// TIA Portal V20 export
FUNCTION_BLOCK "FB_PartControl"   // FB58, SCL
{ S7_Optimized_Access := 'TRUE' }
// stored: MemoryReserve 100, SetENOAutomatically false
   VAR_INPUT
      iStartSeqCond : Bool;   // Start Sequence Conditions
      iJobReq : Bool;   // Job Request - From Main
      iCtrlEnabled : Bool;   // Part Control Enable - Param or Condition
      iShuttleCtrlUndrilledPos : Bool;   // Undrilled Pos. Reached (Option Individual Ctrl) - Param
      iShuttleCtrlUndrilledPosSetPoint : LReal;   // Undrilled Pos. Setpoint (Option Individual Ctrl) - Param
      iShuttleCtrlDrilledPos : Bool;   // Drilled Pos. Reached (Option Individual Ctrl) - Param
      iShuttleCtrlDrilledPosSetPoint : LReal;   // Drilled Pos. Setpoint (Option Individual Ctrl) - Param
      iShuttleCtrlPos : Bool;   // Control Pos. Reached (Option Common Ctrl) - Param
      iShuttleCtrlPosSetPoint : LReal;   // Control Pos. Setpoint (Option Common Ctrl) - Param
      iExpectedCtrlUndrilled : Bool;   // Expected result Undrilled Pos.
      iExpectedCtrlDrilled : Bool;   // Expected result Drilled Pos.
      iPartMeasureValue : Real;   // Part Measure Value (Option Analog Measure) - From AI
      iPartMeasureTolMin : Real;   // Part Tol Min Value (Option Analog Measure) - Param
      iPartMeasureTolMax : Real;   // Part Tol Max Value (Option Analog Measure) - Param
      iUndrilledPartPresence : Bool;
      iDrilledPartPresence : Bool;
      iShuttleMoving : Bool;   // Shuttle is moving - From FB_LoaderAxis
      iShuttleInPos : Bool;   // Shuttle pos. reached - From FB_LoaderAxis
      iPLC_DateAndTime : DTL;
      iStepPause : Bool;
   END_VAR
   VAR_OUTPUT
      oShuttleStartReq { ExternalAccessible := 'False'; ExternalVisible := 'False'; ExternalWritable := 'False'} : Bool;   // Shuttle Start Order - To FB_LoaderAxis
      oShuttlePosSetPoint { ExternalAccessible := 'False'; ExternalVisible := 'False'; ExternalWritable := 'False'} : Real;   // Shuttle Position Setpoint - To FB_LoaderAxis
      oPartControlOK : Bool;   // Part OK - To Main
      oPartControlNOK : Bool;   // Part NOK - To Main
   END_VAR
   VAR
      sCurrent_Step_NB : Int;   // Active Step Number
      sCheck_Step_Condition : Bool;
      sOneStepForward : Bool;
      sRTOneStepForward : R_TRIG;
      sOneStepMode { S7_SetPoint := 'True'} : Bool;
      sStepForward : Bool;
      sInterface : "UDT_SequenceInterface";
      sShuttleStartReq { ExternalAccessible := 'False'; ExternalVisible := 'False'; ExternalWritable := 'False'} : Bool;
      sShuttlePosSetPoint { ExternalAccessible := 'False'; ExternalVisible := 'False'; ExternalWritable := 'False'} : Real;
      sMissingPartCtrlUndrilled : Bool;
      sMissingPartCtrlDrilled : Bool;
      sExtraPartCtrlUndrilled : Bool;
      sExtraPartCtrlDrilled : Bool;
      sPresencePartUndrilledPos : Bool;
      sPresencePartDrilledPos : Bool;
      sPartControlOK : Bool;
      sPartControlNOK : Bool;
      sControlTimer : TON_TIME;
      sHistory : Struct
         Activation : Bool;
         Steps : Array[0..99] of Int;
         Date_Time : Array[0..99] of DTL;
      END_STRUCT;
      StepText : "FB_GetTextErrorCode";
   END_VAR
   VAR_TEMP
      tIndex : Int;   // Index
   END_VAR
   VAR CONSTANT
      S00_INIT : Int := 0;
      S10_CHECK_PART_PRESENCE_OPTION : Int := 10;
      S20_SHUTTLE_TO_UNDRILLED_POS_START_REQ : Int := 20;
      S30_SHUTTLE_TO_UNDRILLED_POS_REACHED : Int := 30;
      S40_WAIT_UNDRILLED_CTRL_EXECUTION : Int := 40;
      S50_SHUTTLE_TO_DRILLED_POS_START_REQ : Int := 50;
      S60_SHUTTLE_TO_DRILLED_POS_REACHED : Int := 60;
      S70_WAIT_DRILLED_CTRL_EXECUTION : Int := 70;
      S80_CHECK_PART_POS_RESULT : Int := 80;
      S120_SHUTTLE_TO_CONTROL_POS_START_REQ : Int := 120;
      S130_SHUTTLE_TO_CONTROL_POS_REACHED : Int := 130;
      S140_WAIT_CONTROL_EXECUTION : Int := 140;
      S180_CHECK_PART_POS_RESULT : Int := 180;
      S280_NO_PART_CTRL : Int := 280;
      S295_JOB_DONE : Int := 295;
   END_VAR
   // StepText.sCode_error[0].ErrorCode := 0;
   // StepText.sCode_error[1].ErrorCode := 10;
   // StepText.sCode_error[2].ErrorCode := 20;
   // StepText.sCode_error[3].ErrorCode := 30;
   // StepText.sCode_error[4].ErrorCode := 40;
   // StepText.sCode_error[5].ErrorCode := 50;
   // StepText.sCode_error[6].ErrorCode := 60;
   // StepText.sCode_error[7].ErrorCode := 70;
   // StepText.sCode_error[8].ErrorCode := 80;
   // StepText.sCode_error[9].ErrorCode := 90;
   // StepText.sCode_error[10].ErrorCode := 95;
BEGIN
   REGION Description header 
       //==================================================================================
       // POSALUX Swiss SA / (C) Copyright 2025
       //----------------------------------------------------------------------------------
       // Title: FB_PartControl
       // Comment/Function: 
       // Author: Fabien WALDT
       // Engineering: TIA Portal v17
       //----------------------------------------------------------------------------------
       // Change log table:
       // Version  | Date     | Expert in charge | Changes applied
       // ---------|----------|------------------|-----------------------------------------
       // 00.00.01 | 20250527 | WFA              | First released version
       // =================================================================================
   END_REGION

   REGION Define condition to start
       IF #iStartSeqCond THEN
           #sInterface.SequenceReleased := TRUE;
       ELSE
           // Standard sequencer controls
           #sInterface.SequenceReleased := FALSE;
           #sCurrent_Step_NB := #S00_INIT;
           #sInterface.SequenceRun := FALSE;
           #sInterface.JobDone := FALSE;
           #sCheck_Step_Condition := FALSE;

           // Dedicated sequencer controls
           #sShuttleStartReq := FALSE;
           #sShuttlePosSetPoint := 0.0;
           #sPresencePartUndrilledPos := FALSE;
           #sPresencePartDrilledPos := FALSE;

           // Add specifics controls 
       END_IF;

       // Reset interface error
       IF #sInterface.Reset THEN
           #sInterface.Error := FALSE;
       END_IF;

       // Reset start when axis in position
       IF #iShuttleInPos THEN
           #sShuttleStartReq := FALSE;
       END_IF;

       // One step forward
       #sRTOneStepForward.CLK := #sOneStepForward;
       #sRTOneStepForward();
       #sStepForward := (NOT #sOneStepMode OR (#sOneStepMode AND #sRTOneStepForward.Q)) AND NOT #iStepPause;
       #sOneStepForward := FALSE;

       // Step Timer
       #sControlTimer(IN := #sCurrent_Step_NB = 40 OR #sCurrent_Step_NB = 140,
                            PT := T#50ms);
   END_REGION

   REGION Sequence Function
       CASE #sCurrent_Step_NB OF
           #S00_INIT:
               REGION S00 INIT
                   #sCheck_Step_Condition := TRUE;
               END_REGION
           #S10_CHECK_PART_PRESENCE_OPTION:
               REGION S10_CHECK_PART_PRESENCE_OPTION
                   #sPartControlOK := FALSE;
                   #sPartControlNOK := FALSE;
                   #sMissingPartCtrlUndrilled := FALSE;
                   #sMissingPartCtrlDrilled := FALSE;
                   #sExtraPartCtrlUndrilled := FALSE;
                   #sExtraPartCtrlDrilled := FALSE;
                   #sCheck_Step_Condition := TRUE;
               END_REGION
           #S20_SHUTTLE_TO_UNDRILLED_POS_START_REQ:
               REGION S20_SHUTTLE_TO_UNDRILLED_POS_START_REQ
                   #sShuttleStartReq := NOT #iShuttleCtrlUndrilledPos;
                   #sShuttlePosSetPoint := LREAL_TO_REAL(#iShuttleCtrlUndrilledPosSetPoint);
                   #sCheck_Step_Condition := TRUE;
               END_REGION
           #S30_SHUTTLE_TO_UNDRILLED_POS_REACHED:
               REGION S30_SHUTTLE_TO_UNDRILLED_POS_REACHED
                   #sCheck_Step_Condition := TRUE;
               END_REGION
           #S40_WAIT_UNDRILLED_CTRL_EXECUTION:
               REGION S40_WAIT_UNDRILLED_CTRL_EXECUTION
                   IF "DB_LoaderOptions".PartControl.AnalogMeasure THEN
                       IF #iPartMeasureValue > #iPartMeasureTolMin AND #iPartMeasureValue < #iPartMeasureTolMax THEN
                           #sPresencePartUndrilledPos := TRUE;
                       ELSE
                           #sPresencePartUndrilledPos := FALSE;
                       END_IF;
                   ELSIF "DB_LoaderOptions".PartControl.DigitalMeasure THEN
                       IF #iUndrilledPartPresence THEN
                           #sPresencePartUndrilledPos := TRUE;
                       ELSE
                           #sPresencePartUndrilledPos := FALSE;
                       END_IF;
                       IF #iDrilledPartPresence THEN
                           #sPresencePartDrilledPos := TRUE;
                       ELSE
                           #sPresencePartDrilledPos := FALSE;
                       END_IF;
                   ELSE
                       #sInterface.Error := TRUE;
                   END_IF;
                   IF #sControlTimer.Q THEN
                       #sCheck_Step_Condition := TRUE;
                   END_IF;
               END_REGION
           #S50_SHUTTLE_TO_DRILLED_POS_START_REQ:
               REGION S50_SHUTTLE_TO_DRILLED_POS_START_REQ
                   #sShuttleStartReq := NOT #iShuttleCtrlDrilledPos;
                   #sShuttlePosSetPoint := LREAL_TO_REAL(#iShuttleCtrlDrilledPosSetPoint);
                   #sCheck_Step_Condition := TRUE;
               END_REGION
           #S60_SHUTTLE_TO_DRILLED_POS_REACHED:
               REGION S60_SHUTTLE_TO_DRILLED_POS_REACHED
                   #sCheck_Step_Condition := TRUE;
               END_REGION
           #S70_WAIT_DRILLED_CTRL_EXECUTION:
               REGION S70_WAIT_DRILLED_CTRL_EXECUTION
                   IF "DB_LoaderOptions".PartControl.AnalogMeasure THEN
                       IF #iPartMeasureValue > #iPartMeasureTolMin AND #iPartMeasureValue < #iPartMeasureTolMax THEN
                           #sPresencePartUndrilledPos := TRUE;
                       ELSE
                           #sPresencePartUndrilledPos := FALSE;
                       END_IF;
                   ELSIF "DB_LoaderOptions".PartControl.DigitalMeasure THEN
                       IF #iUndrilledPartPresence THEN
                           #sPresencePartUndrilledPos := TRUE;
                       ELSE
                           #sPresencePartUndrilledPos := FALSE;
                       END_IF;
                   ELSE
                       #sInterface.Error := TRUE;
                   END_IF;
                   #sCheck_Step_Condition := TRUE;
               END_REGION
           #S80_CHECK_PART_POS_RESULT:
               REGION S80_CHECK_PART_POS_RESULT
                   #sExtraPartCtrlUndrilled := #sPresencePartUndrilledPos AND NOT #iExpectedCtrlUndrilled;
                   #sMissingPartCtrlUndrilled := NOT #sPresencePartUndrilledPos AND #iExpectedCtrlUndrilled;
                   #sExtraPartCtrlDrilled := #sPresencePartDrilledPos AND NOT #iExpectedCtrlDrilled;
                   #sMissingPartCtrlDrilled := NOT #sPresencePartDrilledPos AND #iExpectedCtrlDrilled;

                   IF #sPresencePartUndrilledPos = #iExpectedCtrlUndrilled AND #sPresencePartDrilledPos = #iExpectedCtrlDrilled THEN
                       #sPartControlOK := TRUE;
                       #sPartControlNOK := FALSE;
                   ELSE
                       #sPartControlOK := FALSE;
                       #sPartControlNOK := TRUE;
                   END_IF;
                   #sCheck_Step_Condition := TRUE;
               END_REGION

           #S120_SHUTTLE_TO_CONTROL_POS_START_REQ:
               REGION S120_SHUTTLE_TO_CONTROL_POS_START_REQ
                   #sShuttleStartReq := NOT #iShuttleCtrlPos;
                   #sShuttlePosSetPoint := LREAL_TO_REAL(#iShuttleCtrlPosSetPoint);
                   #sCheck_Step_Condition := TRUE;
               END_REGION
           #S130_SHUTTLE_TO_CONTROL_POS_REACHED:
               REGION S130_SHUTTLE_TO_CONTROL_POS_REACHED
                   #sCheck_Step_Condition := TRUE;
               END_REGION
           #S140_WAIT_CONTROL_EXECUTION:
               REGION S140_WAIT_CONTROL_EXECUTION
                   IF "DB_LoaderOptions".PartControl.AnalogMeasure THEN
                       IF #iPartMeasureValue > #iPartMeasureTolMin AND #iPartMeasureValue < #iPartMeasureTolMax THEN
                           #sPresencePartUndrilledPos := TRUE;
                       ELSE
                           #sPresencePartUndrilledPos := FALSE;
                       END_IF;
                   ELSIF "DB_LoaderOptions".PartControl.DigitalMeasure THEN
                       IF #iUndrilledPartPresence THEN
                           #sPresencePartUndrilledPos := TRUE;
                       ELSE
                           #sPresencePartUndrilledPos := FALSE;
                       END_IF;
                       IF #iDrilledPartPresence THEN
                           #sPresencePartDrilledPos := TRUE;
                       ELSE
                           #sPresencePartDrilledPos := FALSE;
                       END_IF;
                   ELSE
                       #sInterface.Error := TRUE;
                   END_IF;
                   IF #sControlTimer.Q THEN
                       #sCheck_Step_Condition := TRUE;
                   END_IF;
               END_REGION
           #S180_CHECK_PART_POS_RESULT:
               REGION S180_CHECK_PART_POS_RESULT
                   #sExtraPartCtrlUndrilled := #sPresencePartUndrilledPos AND NOT #iExpectedCtrlUndrilled;
                   #sMissingPartCtrlUndrilled := NOT #sPresencePartUndrilledPos AND #iExpectedCtrlUndrilled;
                   #sExtraPartCtrlDrilled := #sPresencePartDrilledPos AND NOT #iExpectedCtrlDrilled;
                   #sMissingPartCtrlDrilled := NOT #sPresencePartDrilledPos AND #iExpectedCtrlDrilled;

                   IF #sPresencePartUndrilledPos = #iExpectedCtrlUndrilled AND #sPresencePartDrilledPos = #iExpectedCtrlDrilled THEN
                       #sPartControlOK := TRUE;
                       #sPartControlNOK := FALSE;
                   ELSE
                       #sPartControlOK := FALSE;
                       #sPartControlNOK := TRUE;
                   END_IF;
                   #sCheck_Step_Condition := TRUE;
               END_REGION

           #S280_NO_PART_CTRL:
               REGION S280_NO_PART_CTRL
                   #sPartControlOK := TRUE;
                   #sPartControlNOK := FALSE;
                   #sCheck_Step_Condition := TRUE;
               END_REGION

           #S295_JOB_DONE:
               REGION S295_JOB_DONE
                   #sInterface.JobDone := TRUE;
                   #sCheck_Step_Condition := TRUE;
               END_REGION
           ELSE:
               #sInterface.Error := TRUE;
       END_CASE;
   END_REGION

   REGION Sequence Next Step Condition
       IF #sCheck_Step_Condition THEN
           CASE #sCurrent_Step_NB OF
               #S00_INIT:
                   REGION S00 INIT
                       IF #sInterface.SequenceReleased AND #iJobReq THEN
                           #sCurrent_Step_NB := #S10_CHECK_PART_PRESENCE_OPTION;
                           #sInterface.SequenceRun := TRUE;
                           #sCheck_Step_Condition := FALSE;
                       ELSE
                           #sInterface.SequenceRun := FALSE;
                       END_IF;
                   END_REGION
               #S10_CHECK_PART_PRESENCE_OPTION:
                   REGION S10_CHECK_PART_PRESENCE_OPTION
                       IF #sInterface.SequenceReleased AND #sStepForward AND "DB_LoaderOptions".PartControl.Individual AND (NOT "DB_LoaderOptions".PartControl.Disabled AND #iCtrlEnabled) THEN
                           #sCurrent_Step_NB := #S20_SHUTTLE_TO_UNDRILLED_POS_START_REQ;
                           #sCheck_Step_Condition := FALSE;
                       ELSIF #sInterface.SequenceReleased AND #sStepForward AND "DB_LoaderOptions".PartControl.Common AND (NOT "DB_LoaderOptions".PartControl.Disabled AND #iCtrlEnabled) THEN
                           #sCurrent_Step_NB := #S120_SHUTTLE_TO_CONTROL_POS_START_REQ;
                           #sCheck_Step_Condition := FALSE;
                       ELSIF #sInterface.SequenceReleased AND #sStepForward AND ("DB_LoaderOptions".PartControl.Disabled OR NOT #iCtrlEnabled) THEN
                           #sCurrent_Step_NB := #S280_NO_PART_CTRL;
                           #sCheck_Step_Condition := FALSE;
                       END_IF;
                   END_REGION
               #S20_SHUTTLE_TO_UNDRILLED_POS_START_REQ:
                   REGION S20_SHUTTLE_TO_UNDRILLED_POS_START_REQ
                       IF #sInterface.SequenceReleased AND (#iShuttleMoving OR #iShuttleCtrlUndrilledPos) THEN
                           #sCurrent_Step_NB := #S30_SHUTTLE_TO_UNDRILLED_POS_REACHED;
                           #sCheck_Step_Condition := FALSE;
                       END_IF;
                   END_REGION
               #S30_SHUTTLE_TO_UNDRILLED_POS_REACHED:
                   REGION S30_SHUTTLE_TO_UNDRILLED_POS_REACHED
                       IF #sInterface.SequenceReleased AND #sStepForward AND NOT #sShuttleStartReq AND #iShuttleCtrlUndrilledPos THEN
                           #sCurrent_Step_NB := #S40_WAIT_UNDRILLED_CTRL_EXECUTION;
                           #sCheck_Step_Condition := FALSE;
                       END_IF;
                   END_REGION
               #S40_WAIT_UNDRILLED_CTRL_EXECUTION:
                   REGION S40_WAIT_UNDRILLED_CTRL_EXECUTION
                       IF #sInterface.SequenceReleased AND #sStepForward AND "AlwaysTRUE" THEN
                           #sCurrent_Step_NB := #S50_SHUTTLE_TO_DRILLED_POS_START_REQ;
                           #sCheck_Step_Condition := FALSE;
                       END_IF;
                   END_REGION
               #S50_SHUTTLE_TO_DRILLED_POS_START_REQ:
                   REGION S50_SHUTTLE_TO_DRILLED_POS_START_REQ
                       IF #sInterface.SequenceReleased AND (#iShuttleMoving OR #iShuttleCtrlDrilledPos) THEN
                           #sCurrent_Step_NB := #S60_SHUTTLE_TO_DRILLED_POS_REACHED;
                           #sCheck_Step_Condition := FALSE;
                       END_IF;
                   END_REGION
               #S60_SHUTTLE_TO_DRILLED_POS_REACHED:
                   REGION S60_SHUTTLE_TO_DRILLED_POS_REACHED
                       IF #sInterface.SequenceReleased AND #sStepForward AND NOT #sShuttleStartReq AND #iShuttleCtrlDrilledPos THEN
                           #sCurrent_Step_NB := #S70_WAIT_DRILLED_CTRL_EXECUTION;
                           #sCheck_Step_Condition := FALSE;
                       END_IF;
                   END_REGION
               #S70_WAIT_DRILLED_CTRL_EXECUTION:
                   REGION S70_WAIT_DRILLED_CTRL_EXECUTION
                       IF #sInterface.SequenceReleased AND #sStepForward AND "AlwaysTRUE" THEN
                           #sCurrent_Step_NB := #S80_CHECK_PART_POS_RESULT;
                           #sCheck_Step_Condition := FALSE;
                       END_IF;
                   END_REGION
               #S80_CHECK_PART_POS_RESULT:
                   REGION S80_CHECK_PART_POS_RESULT
                       IF #sInterface.SequenceReleased AND #sStepForward AND "AlwaysTRUE" THEN
                           #sCurrent_Step_NB := #S295_JOB_DONE;
                           #sCheck_Step_Condition := FALSE;
                       END_IF;
                   END_REGION

               #S120_SHUTTLE_TO_CONTROL_POS_START_REQ:
                   REGION S120_SHUTTLE_TO_CONTROL_POS_START_REQ
                       IF #sInterface.SequenceReleased AND (#iShuttleMoving OR #iShuttleCtrlPos) THEN
                           #sCurrent_Step_NB := #S130_SHUTTLE_TO_CONTROL_POS_REACHED;
                           #sCheck_Step_Condition := FALSE;
                       END_IF;
                   END_REGION
               #S130_SHUTTLE_TO_CONTROL_POS_REACHED:
                   REGION S130_SHUTTLE_TO_CONTROL_POS_REACHED
                       IF #sInterface.SequenceReleased AND #sStepForward AND NOT #sShuttleStartReq AND #iShuttleCtrlPos THEN
                           #sCurrent_Step_NB := #S140_WAIT_CONTROL_EXECUTION;
                           #sCheck_Step_Condition := FALSE;
                       END_IF;
                   END_REGION
               #S140_WAIT_CONTROL_EXECUTION:
                   REGION S140_WAIT_CONTROL_EXECUTION
                       IF #sInterface.SequenceReleased AND #sStepForward AND "AlwaysTRUE" THEN
                           #sCurrent_Step_NB := #S180_CHECK_PART_POS_RESULT;
                           #sCheck_Step_Condition := FALSE;
                       END_IF;
                   END_REGION
               #S180_CHECK_PART_POS_RESULT:
                   REGION S180_CHECK_PART_POS_RESULT
                       IF #sInterface.SequenceReleased AND #sStepForward AND "AlwaysTRUE" THEN
                           #sCurrent_Step_NB := #S295_JOB_DONE;
                           #sCheck_Step_Condition := FALSE;
                       END_IF;
                   END_REGION

               #S280_NO_PART_CTRL:
                   REGION S280_NO_PART_CTRL
                       IF #sInterface.SequenceReleased AND #sStepForward AND "AlwaysTRUE" THEN
                           #sCurrent_Step_NB := #S295_JOB_DONE;
                           #sCheck_Step_Condition := FALSE;
                       END_IF;
                   END_REGION

               #S295_JOB_DONE:
                   REGION S95_JOB_DONE
                       IF NOT #iJobReq THEN
                           #sCurrent_Step_NB := #S00_INIT;
                           #sCheck_Step_Condition := FALSE;
                           #sInterface.JobDone := FALSE;
                       END_IF;
                   END_REGION
               ELSE
                   #sInterface.Error := TRUE;
           END_CASE;
       END_IF;
   END_REGION

   REGION Outputs Update
       #oShuttleStartReq := #sShuttleStartReq;
       #oShuttlePosSetPoint:= #sShuttlePosSetPoint;
       #oPartControlOK := #sPartControlOK;
       #oPartControlNOK := #sPartControlNOK;
   END_REGION

   REGION Steps - Date and Time History
       IF #sHistory.Activation THEN
           IF #sHistory.Steps[0] <> #sCurrent_Step_NB THEN
               FOR #tIndex := 98 TO 0 BY -1 DO
                   #sHistory.Steps[#tIndex + 1] := #sHistory.Steps[#tIndex];
                   #sHistory.Date_Time[#tIndex + 1] := #sHistory.Date_Time[#tIndex];
               END_FOR;
               #sHistory.Steps[0] := #sCurrent_Step_NB;
               #sHistory.Date_Time[0] := #iPLC_DateAndTime;
           END_IF;
       END_IF;
   END_REGION

   REGION Steps Text
       #StepText(iErrorCode := #sCurrent_Step_NB,
                 oErrorText => #StepText.oErrorText);
   END_REGION
END_FUNCTION_BLOCK
